Fanuc KAREL source: kt00751.KL

-- PROVISIONAL review KL for V770-1; original PC SHA256 6508fac8cfa98d9a3d0ec7a00bf50af6a175a70f99825d5503dfb787abe291c5
-- Incomplete behavior may be omitted. Consult companion uncertainty JSON. Do not deploy.
PROGRAM KT00751
%NOLOCKGROUP
VAR
  R1 : REAL
  R2 : REAL
  OUT : REAL
BEGIN
  -- UNRESOLVED_PC offsets 5-16; opcodes 2E,23
  -- UNRESOLVED_PC offsets 21-32; opcodes 2E,23
  -- UNRESOLVED_PC offsets 37-48; opcodes 2E,23
  -- UNRESOLVED_PC offsets 53-64; opcodes 2E,23
  -- UNRESOLVED_PC offsets 69-82; opcodes 21,67,23
  -- UNRESOLVED_PC offsets 87-91; opcodes 7F
END KT00751
